PROGRAM PRG_1_PlcTask
VAR

END_VAR

PRG_MR1K2();
//PRG_SP1K1_MONO();

END_PROGRAM

(* stored: Version 1.1.0.1, ProductVersion 3.1.4022.18
   POU PRG_1_PlcTask: Id {21f3a158-4837-47ff-8ec7-29454a44967d}, SpecialFunc None *)
